// TIA Portal V17 export
// export: Created 2025-03-07T09:19:07.1969303Z, ExportSetting WithDefaults, DisplayName Totally Integrated Automation Portal, DisplayVersion V17 Update 8, DisplayName TIA Portal Openness, DisplayVersion V17 Update 8, DisplayName TIA Portal Version Control Interface, DisplayVersion V17, DisplayName SINAMICS Startdrive Advanced, DisplayVersion V17 SP2, DisplayName SINAMICS Startdrive G110M, G120, G120C, G120D, G120P, G115D, DisplayVersion V17 SP2, DisplayName SINAMICS Startdrive G130, G150, S120, S150, SINAMICS MV, S210, DisplayVersion V17 SP2, DisplayName STEP 7 Professional, DisplayVersion V17 Update 8, DisplayName SINUMERIK ONE STEP 7 Toolbox, DisplayVersion V17 Update 12, DisplayName SINUMERIK 840D sl STEP 7 Toolbox, DisplayVersion V17 Update 12, DisplayName STEP 7 Safety, DisplayVersion V17 Update 6, DisplayName WinCC Advanced, DisplayVersion V17 Update 8
FUNCTION_BLOCK "FB10101_POWDER_FLOW_SENSOR_MEDICOAT"   // FB10101, LAD
{ S7_Optimized_Access := 'FALSE' }
VERSION : 0.1
// stored: AutoNumber false, IsIECCheckEnabled false, SetENOAutomatically false, UDAEnableTagReadback false
   VAR_INPUT
      ANALOG_VALUE : Int;   // SENSOR VALUE INPUT
      UNIT_NO : Int;   // UNIT NUMBER
      TIMER_1 : Timer;   // TIMER FOR NOT FLOW ALARM
      POWDER_FEEDER_ON { ExternalVisible := 'False'; ExternalWritable := 'False'} : Bool;   // POWDER FEEDER SWITCHED ON
   END_VAR
   VAR_OUTPUT
      POWDER_FLOW_ON : Bool;   // POWDER FLOW OK
      NO_POWDER_FLOW_ALARM : Bool;   // NO POWDER FLOW ALARM
      WARNING_LIMIT : Bool;   // WARNING FLOW OUT OF LIMITS
      ERROR_CONFIGURATION : Bool;   // WRONG CONFIGURATION ERROR
   END_VAR
   VAR DB_SPECIFIC
      OUTPUT : Struct
         VALUE_REAL : Real;   // POWDER FLOW VALUE
         VALUE_INT : Int;
      END_STRUCT;
      INPUT_SETTINGS : Struct
         LOW_RANGE : Real;   // LOWER VALUE TO SCALE ANALOG SIGNAL
         HIGH_RANGE : Real;   // HIGHER VALUE TO SCALE ANALOG SIGNAL
         LOW_LIMIT_TO_POWDER_FLOW_ON : Real;   // MINIMUM VALUE TO POWDER FLOW OK
      END_STRUCT;
      ALARMS_SETTINGS : Struct
         WARN_LIMIT_LOW : Real;   // LOWER LIMIT FOR WARNING
         WARN_LIMIT_HIGH : Real;   // HIGHER LIMIT FOR WARNING
      END_STRUCT;
      LOG : Struct
         DATE_MAX_MASS : Date_And_Time;
         VALUE_MAX_MASS : Real;
      END_STRUCT;
      INPUT_DINT : DInt;   // SENSOR VALUE INPUT DINT
   END_VAR
   VAR_TEMP
      NORM_VALUE : Real;
      RETVAL : Word;
   END_VAR
   VAR CONSTANT
      FB_NUMBER : DInt := 21200;
   END_VAR
   VAR_TEMP   // added for the SCL form of the ladder/FBD networks
      _w1 : Bool;
      _s5time1 : S5Time;
   END_VAR
BEGIN

REGION Network 1: INPUTS
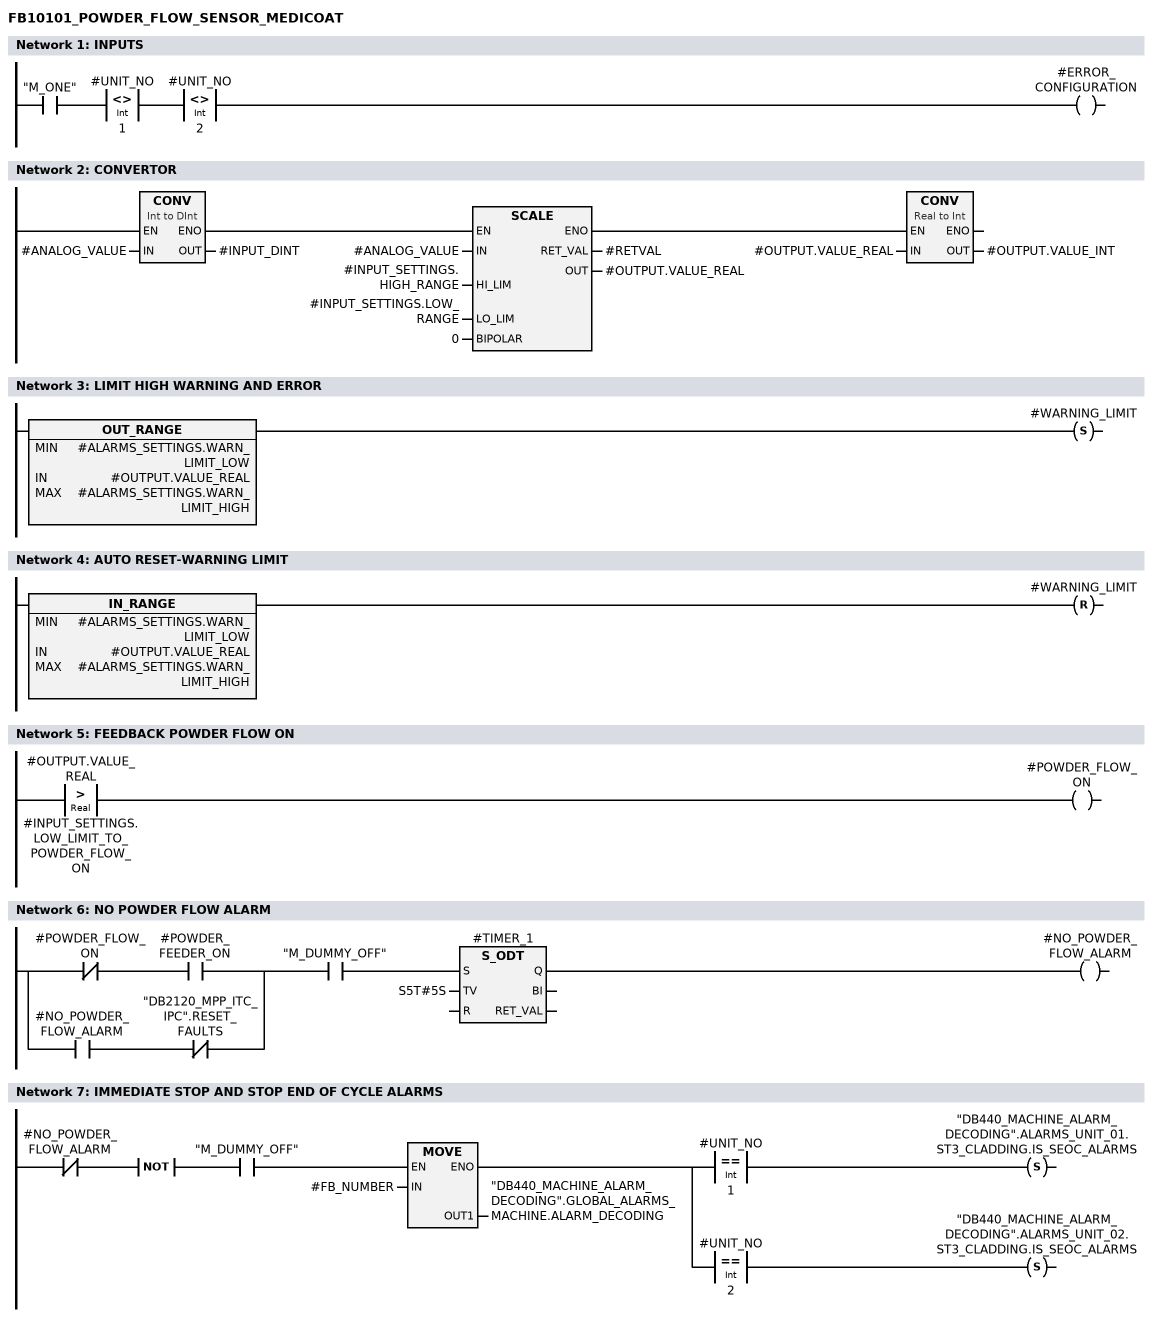
   RUNG wire#powerrail
      Contact( "M_ONE" )
      { S7_Templates := "SrcType := Int" } NE_Contact(in1 := #UNIT_NO, in2 := 1)
      { S7_Templates := "SrcType := Int" } NE_Contact(in1 := #UNIT_NO, in2 := 2)
      Coil( #ERROR_CONFIGURATION )
   END_RUNG
   // the same network as SCL:
   #ERROR_CONFIGURATION := "M_ONE" AND (#UNIT_NO <> 1) AND (#UNIT_NO <> 2);
END_REGION

REGION Network 2: CONVERTOR
   #INPUT_DINT := INT_TO_DINT(#ANALOG_VALUE);
   #RETVAL := SCALE(IN := #ANALOG_VALUE,
                    HI_LIM := #INPUT_SETTINGS.HIGH_RANGE,
                    LO_LIM := #INPUT_SETTINGS.LOW_RANGE,
                    BIPOLAR := 0,
                    OUT => #OUTPUT.VALUE_REAL,
                    ENO => #_w1);
   IF #_w1 THEN #OUTPUT.VALUE_INT := REAL_TO_INT(#OUTPUT.VALUE_REAL); END_IF;
END_REGION

REGION Network 3: LIMIT HIGH WARNING AND ERROR
   IF (#OUTPUT.VALUE_REAL < #ALARMS_SETTINGS.WARN_LIMIT_LOW) OR (#OUTPUT.VALUE_REAL > #ALARMS_SETTINGS.WARN_LIMIT_HIGH) THEN
       #WARNING_LIMIT := TRUE;
   END_IF;
END_REGION

REGION Network 4: AUTO RESET-WARNING LIMIT
   RUNG wire#powerrail
      { S7_Templates := "SrcType := Real" } InRange(min := #ALARMS_SETTINGS.WARN_LIMIT_LOW, in := #OUTPUT.VALUE_REAL, max := #ALARMS_SETTINGS.WARN_LIMIT_HIGH)
      R_Coil( #WARNING_LIMIT )
   END_RUNG
   // the same network as SCL:
   IF (#ALARMS_SETTINGS.WARN_LIMIT_LOW <= #OUTPUT.VALUE_REAL) AND (#OUTPUT.VALUE_REAL <= #ALARMS_SETTINGS.WARN_LIMIT_HIGH) THEN
       #WARNING_LIMIT := FALSE;
   END_IF;
END_REGION

REGION Network 5: FEEDBACK POWDER FLOW ON
   RUNG wire#powerrail
      { S7_Templates := "SrcType := Real" } GT_Contact(in1 := #OUTPUT.VALUE_REAL, in2 := #INPUT_SETTINGS.LOW_LIMIT_TO_POWDER_FLOW_ON)
      Coil( #POWDER_FLOW_ON )
   END_RUNG
   // the same network as SCL:
   #POWDER_FLOW_ON := #OUTPUT.VALUE_REAL > #INPUT_SETTINGS.LOW_LIMIT_TO_POWDER_FLOW_ON;
END_REGION

REGION Network 6: NO POWDER FLOW ALARM
   RUNG wire#powerrail
      I_Contact( #POWDER_FLOW_ON )
      Contact( #POWDER_FEEDER_ON )
      wire#w1
      Contact( "M_DUMMY_OFF" )
      S_ODT(T_NO := #TIMER_1, TV := S5T#5S, R :=, BI =>, RET_VAL =>)
      Coil( #NO_POWDER_FLOW_ALARM )
   END_RUNG
   RUNG wire#powerrail
      Contact( #NO_POWDER_FLOW_ALARM )
      I_Contact( "DB2120_MPP_ITC_IPC".RESET_FAULTS )
   END_RUNG wire#w1
   // the same network as SCL:
   #_s5time1 := S_ODT(T_NO := #TIMER_1,
                      S := ((NOT #POWDER_FLOW_ON AND #POWDER_FEEDER_ON) OR (#NO_POWDER_FLOW_ALARM AND NOT "DB2120_MPP_ITC_IPC".RESET_FAULTS)) AND "M_DUMMY_OFF",
                      TV := S5T#5S,
                      Q => #_w1);
   #NO_POWDER_FLOW_ALARM := #_w1;
END_REGION

REGION Network 7: IMMEDIATE STOP AND STOP END OF CYCLE ALARMS
   RUNG wire#powerrail
      I_Contact( #NO_POWDER_FLOW_ALARM )
      Not()
      Contact( "M_DUMMY_OFF" )
      Move(in := #FB_NUMBER, out1 => "DB440_MACHINE_ALARM_DECODING".GLOBAL_ALARMS_MACHINE.ALARM_DECODING)
      wire#w1
      { S7_Templates := "SrcType := Int" } EQ_Contact(in1 := #UNIT_NO, in2 := 1)
      S_Coil( "DB440_MACHINE_ALARM_DECODING".ALARMS_UNIT_01.ST3_CLADDING.IS_SEOC_ALARMS )
   END_RUNG
   RUNG wire#w1
      { S7_Templates := "SrcType := Int" } EQ_Contact(in1 := #UNIT_NO, in2 := 2)
      S_Coil( "DB440_MACHINE_ALARM_DECODING".ALARMS_UNIT_02.ST3_CLADDING.IS_SEOC_ALARMS )
   END_RUNG
   // the same network as SCL:
   #_w1 := NOT (NOT #NO_POWDER_FLOW_ALARM) AND "M_DUMMY_OFF";
   IF #_w1 THEN "DB440_MACHINE_ALARM_DECODING".GLOBAL_ALARMS_MACHINE.ALARM_DECODING := #FB_NUMBER; END_IF;
   IF #_w1 AND (#UNIT_NO = 1) THEN
       "DB440_MACHINE_ALARM_DECODING".ALARMS_UNIT_01.ST3_CLADDING.IS_SEOC_ALARMS := TRUE;
   END_IF;
   IF #_w1 AND (#UNIT_NO = 2) THEN
       "DB440_MACHINE_ALARM_DECODING".ALARMS_UNIT_02.ST3_CLADDING.IS_SEOC_ALARMS := TRUE;
   END_IF;
END_REGION
END_FUNCTION_BLOCK
